FUNCTION_BLOCK AR_TO_AR2 (* Composite FB for convert unidirectional AR to bidirectional AR2 *)
  (* Standard: 61499-2; Function: AR_IN publishes its value onto the outgoing (EO1) side of AR2_BIDIR. Whatever AR2_BIDIR receives on its incoming (EI1) side is forwarded out again as a plain unidirectional signal via AR_OUT.; Description: Copyright (c) 2026 HR Agrartechnik GmbH This program and the accompanying materials are made available under the terms of the Eclipse Public License 2.0 which is available at https://www.eclipse.org/legal/epl-2.0/ SPDX-License-Identifier: EPL-2.0 *)
  (* Version 1.0, 2026-08-31, Franz Höpfinger, HR Agrartechnik GmbH, Initial Version *)
  PACKAGE adapter::conversion::bidirectional;
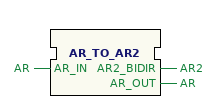
  SOCKETS
    AR_IN : adapter::types::unidirectional::AR; (* Adapter Input: unidirectional source *)
  END_SOCKETS
  PLUGS
    AR2_BIDIR : adapter::types::bidirectional::AR2; (* Adapter Output: bidirectional tap, outgoing side driven by AR_IN, incoming side forwarded to AR_OUT *)
    AR_OUT : adapter::types::unidirectional::AR; (* Adapter Output: mirrors AR2_BIDIR's incoming (request) side *)
  END_PLUGS
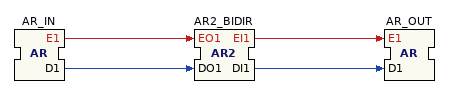
  EVENT_CONNECTIONS
    AR_IN.E1 TO AR2_BIDIR.EO1;
    AR2_BIDIR.EI1 TO AR_OUT.E1;
  END_CONNECTIONS
  DATA_CONNECTIONS
    AR_IN.D1 TO AR2_BIDIR.DO1;
    AR2_BIDIR.DI1 TO AR_OUT.D1;
  END_CONNECTIONS
END_FUNCTION_BLOCK
